TYPE E_MainStep :
(
	ePREPARE_SUBSCRIPTION := 0,
	ePREP_PUBLISH,
	ePUBLISH,
	eCHECK_SUBSCRIPTION,
	eEVAL_PAYLOAD,
	ePREPARE_PACKAGE_TIMER 
)UINT;
END_TYPE

(* stored: Version 1.1.0.1, ProductVersion 3.1.4024.2
   DUT E_MainStep: Id {db132ccf-282a-42c2-9dab-7b358aec39c3} *)
